INTERFACE I_HaveOutputPorts EXTENDS __SYSTEM.IQueryInterface

METHOD AddOutputPort
VAR_INPUT
	OutputPortToAdd : I_OutputPort;
END_VAR
END_METHOD

METHOD PUBLIC GetOutputPorts : I_OutputPortCollection
VAR_INPUT
END_VAR
END_METHOD

METHOD PUBLIC TryGetOutputPortByName : BOOL
VAR_INPUT
	Name : T_MAXSTRING;
	Destination : REFERENCE TO I_OutputPort;
END_VAR
END_METHOD

END_INTERFACE

(* stored: Version 1.1.0.1, ProductVersion 3.1.4024.12
   Itf I_HaveOutputPorts: Id {5e1aea97-5e53-08af-11e9-4031292affee}
   Method AddOutputPort: Id {ccc39ff5-e25c-0f20-3efe-f937f75d1bdc}
   Method GetOutputPorts: Id {932c82cf-4cbd-08c5-3c69-c19533529db8}
   Method TryGetOutputPortByName: Id {a3a67671-970b-01d6-2705-151b345eba16} *)
